# EPICS substitutions: apps/xpsMotorApp/Db/XPS3_Aux_ai.substitutions
file "db/XPSAuxAi.db"
{
pattern
{P,          R,          PORT,     CHAN, LOPR,   HOPR,  PREC, SCAN}
{halldxps3:, XPSAuxAi0,  XPS_AUX1, 0,    -10.0,  10.0,  6,    "1 second"}
{halldxps3:, XPSAuxAi1,  XPS_AUX1, 1,    -10.0,  10.0,  6,    "1 second"}
{halldxps3:, XPSAuxAi2,  XPS_AUX1, 2,    -10.0,  10.0,  6,    "1 second"}
{halldxps3:, XPSAuxAi3,  XPS_AUX1, 3,    -10.0,  10.0,  6,    "1 second"}
}
